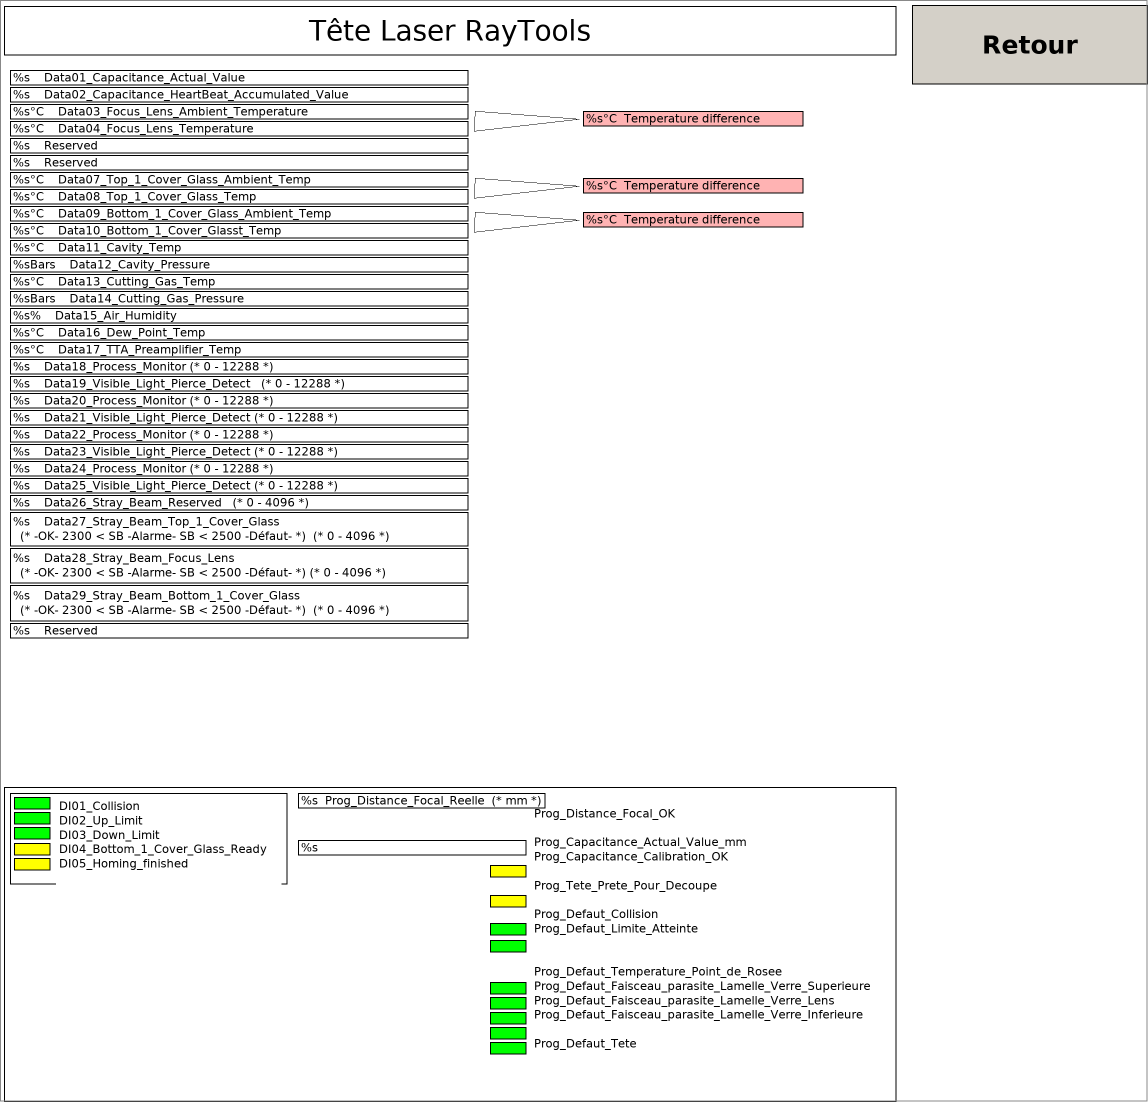
VISUALIZATION Laser_Tete_Raytools_1  // 1148x1102
    Rectangle (583,212 220x15), invisible if: (Data10_Bottom_1_Cover_Glasst_Temp/100) - (Data09_Bottom_1_Cover_Glass_Ambient_Temp/100) >=14
    Rectangle (583,212 220x15), invisible if: (Data10_Bottom_1_Cover_Glasst_Temp/100) - (Data09_Bottom_1_Cover_Glass_Ambient_Temp/100) <14 or (Data10_Bottom_1_Cover_Glasst_Temp/100) - (Data09_Bottom_1_Cover_Glass_Ambient_Temp/100)>=20
    Rectangle (583,212 220x15), invisible if: (Data10_Bottom_1_Cover_Glasst_Temp/100) - (Data09_Bottom_1_Cover_Glass_Ambient_Temp/100) <20
    Rectangle (583,178 220x15), invisible if: (Data08_Top_1_Cover_Glass_Temp/100) - (Data07_Top_1_Cover_Glass_Ambient_Temp/100) >=14
    Rectangle (583,178 220x15), invisible if: (Data08_Top_1_Cover_Glass_Temp/100) - (Data07_Top_1_Cover_Glass_Ambient_Temp/100) <14 or (Data08_Top_1_Cover_Glass_Temp/100) - (Data07_Top_1_Cover_Glass_Ambient_Temp/100)>=20
    Rectangle (583,178 220x15), invisible if: (Data08_Top_1_Cover_Glass_Temp/100) - (Data07_Top_1_Cover_Glass_Ambient_Temp/100) <20
    Rectangle (583,111 220x15), invisible if: (Data04_Focus_Lens_Temperature/100) - (Data03_Focus_Lens_Ambient_Temperature/100) >=14
    Rectangle (583,111 220x15), invisible if: (Data04_Focus_Lens_Temperature/100) - (Data03_Focus_Lens_Ambient_Temperature/100) <14 or (Data04_Focus_Lens_Temperature/100) - (Data03_Focus_Lens_Ambient_Temperature/100)>=20
    Rectangle (583,111 220x15), invisible if: (Data04_Focus_Lens_Temperature/100) - (Data03_Focus_Lens_Ambient_Temperature/100) <20
    Rectangle (10,70 458x15), "%s Data01_Capacitance_Actual_Value", text variable: IO_TETE_LASER_RAYTOOLS.Data01_Capacitance_Actual_Value
    Rectangle (4,787 892x315)
    Rectangle (10,793 277x91)
    Rectangle (14,797 36x12), colour toggle: IO_TETE_LASER_RAYTOOLS.DI01_Collision
    Rectangle (56,798 225x86), "DI01_Collision DI02_Up_Limit DI03_Down_Limit DI04_Bottom_1_Cover_Glass_Ready DI05_Homing_finished"
    Rectangle (14,812 36x12), colour toggle: IO_TETE_LASER_RAYTOOLS.DI02_Up_Limit
    Rectangle (14,827 36x12), colour toggle: IO_TETE_LASER_RAYTOOLS.DI03_Down_Limit
    Rectangle (14,843 36x12), colour toggle: IO_TETE_LASER_RAYTOOLS.DI04_Bottom_1_Cover_Glass_Ready
    Rectangle (14,858 36x12), colour toggle: IO_TETE_LASER_RAYTOOLS.DI05_Homing_finished
    Rectangle (10,87 458x15), "%s Data02_Capacitance_HeartBeat_Accumulated_Value", text variable: IO_TETE_LASER_RAYTOOLS.Data02_Capacitance_HeartBeat_Accumulated_Value
    Rectangle (10,104 458x15), "%s°C Data03_Focus_Lens_Ambient_Temperature", text variable: IO_TETE_LASER_RAYTOOLS.Data03_Focus_Lens_Ambient_Temperature /100
    Rectangle (10,121 458x15), "%s°C Data04_Focus_Lens_Temperature", text variable: IO_TETE_LASER_RAYTOOLS.Data04_Focus_Lens_Temperature /100
    Rectangle (10,138 458x15), "%s Reserved"
    Rectangle (10,155 458x15), "%s Reserved"
    Rectangle (10,172 458x15), "%s°C Data07_Top_1_Cover_Glass_Ambient_Temp", text variable: IO_TETE_LASER_RAYTOOLS.Data07_Top_1_Cover_Glass_Ambient_Temp /100
    Rectangle (10,189 458x15), "%s°C Data08_Top_1_Cover_Glass_Temp", text variable: IO_TETE_LASER_RAYTOOLS.Data08_Top_1_Cover_Glass_Temp
    Rectangle (10,206 458x15), "%s°C Data09_Bottom_1_Cover_Glass_Ambient_Temp", text variable: IO_TETE_LASER_RAYTOOLS.Data09_Bottom_1_Cover_Glass_Ambient_Temp/100
    Rectangle (10,223 458x15), "%s°C Data10_Bottom_1_Cover_Glasst_Temp", text variable: IO_TETE_LASER_RAYTOOLS.Data10_Bottom_1_Cover_Glasst_Temp/100
    Rectangle (10,240 458x15), "%s°C Data11_Cavity_Temp", text variable: IO_TETE_LASER_RAYTOOLS.Data11_Cavity_Temp/100
    Rectangle (10,257 458x15), "%sBars Data12_Cavity_Pressure", text variable: IO_TETE_LASER_RAYTOOLS.Data12_Cavity_Pressure/10
    Rectangle (10,274 458x15), "%s°C Data13_Cutting_Gas_Temp", text variable: IO_TETE_LASER_RAYTOOLS.Data13_Cutting_Gas_Temp/100
    Rectangle (10,291 458x15), "%sBars Data14_Cutting_Gas_Pressure", text variable: IO_TETE_LASER_RAYTOOLS.Data14_Cutting_Gas_Pressure/100
    Rectangle (10,308 458x15), "%s% Data15_Air_Humidity", text variable: IO_TETE_LASER_RAYTOOLS.Data15_Per_10000_Humidity/100
    Rectangle (10,325 458x15), "%s°C Data16_Dew_Point_Temp", text variable: IO_TETE_LASER_RAYTOOLS.Data16_Dew_Point_Temp/100
    Rectangle (10,342 458x15), "%s°C Data17_TTA_Preamplifier_Temp", text variable: IO_TETE_LASER_RAYTOOLS.Data17_TTA_Preamplifier_Temp/100
    Rectangle (10,359 458x15), "%s Data18_Process_Monitor (* 0 - 12288 *)", text variable: IO_TETE_LASER_RAYTOOLS.Data18_Process_Monitor
    Rectangle (10,376 458x15), "%s Data19_Visible_Light_Pierce_Detect (* 0 - 12288 *)", text variable: IO_TETE_LASER_RAYTOOLS.Data19_Visible_Light_Pierce_Detect
    Rectangle (10,393 458x15), "%s Data20_Process_Monitor (* 0 - 12288 *)", text variable: IO_TETE_LASER_RAYTOOLS.Data20_Process_Monitor
    Rectangle (10,410 458x15), "%s Data21_Visible_Light_Pierce_Detect (* 0 - 12288 *)", text variable: IO_TETE_LASER_RAYTOOLS.Data21_Visible_Light_Pierce_Detect
    Rectangle (10,427 458x15), "%s Data22_Process_Monitor (* 0 - 12288 *)", text variable: IO_TETE_LASER_RAYTOOLS.Data22_Process_Monitor
    Rectangle (10,444 458x15), "%s Data23_Visible_Light_Pierce_Detect (* 0 - 12288 *)", text variable: IO_TETE_LASER_RAYTOOLS.Data23_Visible_Light_Pierce_Detect
    Rectangle (10,478 458x15), "%s Data25_Visible_Light_Pierce_Detect (* 0 - 12288 *)", text variable: IO_TETE_LASER_RAYTOOLS.Data25_Visible_Light_Pierce_Detect
    Rectangle (10,495 458x15), "%s Data26_Stray_Beam_Reserved (* 0 - 4096 *)", text variable: IO_TETE_LASER_RAYTOOLS.Data25_Visible_Light_Pierce_Detect
    Rectangle (10,512 458x34), "%s Data27_Stray_Beam_Top_1_Cover_Glass (* -OK- 2300 < SB -Alarme- SB < 2500 -Défaut- *) (* 0 - 4096 *)", text variable: IO_TETE_LASER_RAYTOOLS.Data27_Stray_Beam_Top_1_Cover_Glass
    Rectangle (10,548 458x35), "%s Data28_Stray_Beam_Focus_Lens (* -OK- 2300 < SB -Alarme- SB < 2500 -Défaut- *) (* 0 - 4096 *)", text variable: IO_TETE_LASER_RAYTOOLS.Data28_Stray_Beam_Focus_Lens
    Rectangle (10,585 458x36), "%s Data29_Stray_Beam_Bottom_1_Cover_Glass (* -OK- 2300 < SB -Alarme- SB < 2500 -Défaut- *) (* 0 - 4096 *)", text variable: IO_TETE_LASER_RAYTOOLS.Data29_Stray_Beam_Bottom_1_Cover_Glass
    Rectangle (10,623 458x15), "%s Reserved", text variable: IO_TETE_LASER_RAYTOOLS.Data30_Reserved
    Rectangle (531,791 364x308), "Prog_Distance_Focal_OK Prog_Capacitance_Actual_Value_mm Prog_Capacitance_Calibration_OK Prog_Tete_Prete_Pour_Decoupe Prog_Defaut_Collision Prog_Defaut_Limite_Atteinte Prog_Defaut_Temperature_Point_de_Rosee Prog_Defaut_Faisceau_parasite_Lamelle_Verre_Superieure Prog_Defaut_Faisceau_parasite_Lamelle_Verre_Lens Prog_Defaut_Faisceau_parasite_Lamelle_Verre_Inferieure Prog_Defaut_Tete"
    Rectangle (298,793 247x15), "%s Prog_Distance_Focal_Reelle (* mm *)", text variable: IO_TETE_LASER_RAYTOOLS.Prog_Distance_Focal_Reelle
    Rectangle (298,840 228x15), "%s", text variable: IO_TETE_LASER_RAYTOOLS.Prog_Capacitance_Actual_Value_mm
    Rectangle (490,865 36x12), colour toggle: IO_TETE_LASER_RAYTOOLS.Prog_Capacitance_Calibration_OK
    Rectangle (490,895 36x12), colour toggle: IO_TETE_LASER_RAYTOOLS.Prog_Tete_Prete_Pour_Decoupe
    Rectangle (490,923 36x12), colour toggle: IO_TETE_LASER_RAYTOOLS.Prog_Defaut_Collision
    Rectangle (490,940 36x12), colour toggle: IO_TETE_LASER_RAYTOOLS.Prog_Defaut_Limite_Atteinte
    Rectangle (490,982 36x12), colour toggle: IO_TETE_LASER_RAYTOOLS.Prog_Defaut_Temperature_Lamelle_Verre_Superieure
    Rectangle (490,997 36x12), colour toggle: IO_TETE_LASER_RAYTOOLS.Prog_Defaut_Temperature_Lamelle_Verre_Inferieure
    Rectangle (490,1012 36x12), colour toggle: IO_TETE_LASER_RAYTOOLS.Prog_Defaut_Temperature_Point_de_Rosee
    Rectangle (490,1027 36x12), colour toggle: IO_TETE_LASER_RAYTOOLS.Prog_Defaut_Faisceau_parasite_Lamelle_Verre_Superieure
    Rectangle (490,1042 36x12), colour toggle: IO_TETE_LASER_RAYTOOLS.Prog_Defaut_Faisceau_parasite_Lamelle_Verre_Lens
    Rectangle (4,6 892x49), "Tête Laser RayTools"
    Rectangle (912,5 236x79), "Retour"
        OnMouseClick: change screen: MenuPrincipal
    Rectangle (10,461 458x15), "%s Data24_Process_Monitor (* 0 - 12288 *)", text variable: IO_TETE_LASER_RAYTOOLS.Data24_Process_Monitor
    Rectangle (583,111 220x15), "%s°C Temperature difference", text variable: (IO_TETE_LASER_RAYTOOLS.Data04_Focus_Lens_Temperature /100) - (IO_TETE_LASER_RAYTOOLS.Data03_Focus_Lens_Ambient_Temperature /100)
    Polygon (475,111) (579,119) (474,131)
    Rectangle (583,178 220x15), "%s°C Temperature difference", text variable: (IO_TETE_LASER_RAYTOOLS.Data08_Top_1_Cover_Glass_Temp /100) - (IO_TETE_LASER_RAYTOOLS.Data07_Top_1_Cover_Glass_Ambient_Temp /100)
    Polygon (475,178) (579,186) (474,198)
    Rectangle (583,212 220x15), "%s°C Temperature difference", text variable: (IO_TETE_LASER_RAYTOOLS.Data10_Bottom_1_Cover_Glasst_Temp /100) - (IO_TETE_LASER_RAYTOOLS.Data09_Bottom_1_Cover_Glass_Ambient_Temp /100)
    Polygon (475,212) (579,220) (474,232)
END_VISUALIZATION

(* stored: Version 1.1.0.1
   Visu Laser_Tete_Raytools_1: Id {5736dd0e-5eb8-4b72-b0af-49d39c1c188c} *)
